// TIA Portal V20 export
FUNCTION_BLOCK "LER_EmOverviewHomeCondtion"   // FB182, LAD
// stored: IsIECCheckEnabled true, MemoryReserve 100, Namespace Unit1.Em2, SetENOAutomatically true
   VAR_INPUT
      maxPageCount : Int;
      unitStatus { ExternalAccessible := 'False'; ExternalVisible := 'False'; ExternalWritable := 'False'} : "LAF_typeUnitStatus";   // Current unit status o be used in this EM
   END_VAR
   VAR_IN_OUT
      moduleInterface : "LER_typeEmOverviewHomeCondition";
   END_VAR
   VAR
      statButtonPressedOld : Array[0..1] of Bool;
      statLampControl { ExternalAccessible := 'False'; ExternalVisible := 'False'; ExternalWritable := 'False'} : Bool;
      statPulse { ExternalAccessible := 'False'; ExternalVisible := 'False'; ExternalWritable := 'False'} : Bool;
   END_VAR
   VAR_TEMP
      tempLampOff : Array[0..13] of Bool;
   END_VAR
   VAR_TEMP   // added for the SCL form of the ladder/FBD networks
      _w1 : Bool;
      _w2 : Bool;
   END_VAR
BEGIN

REGION Network 1: Page Index Control
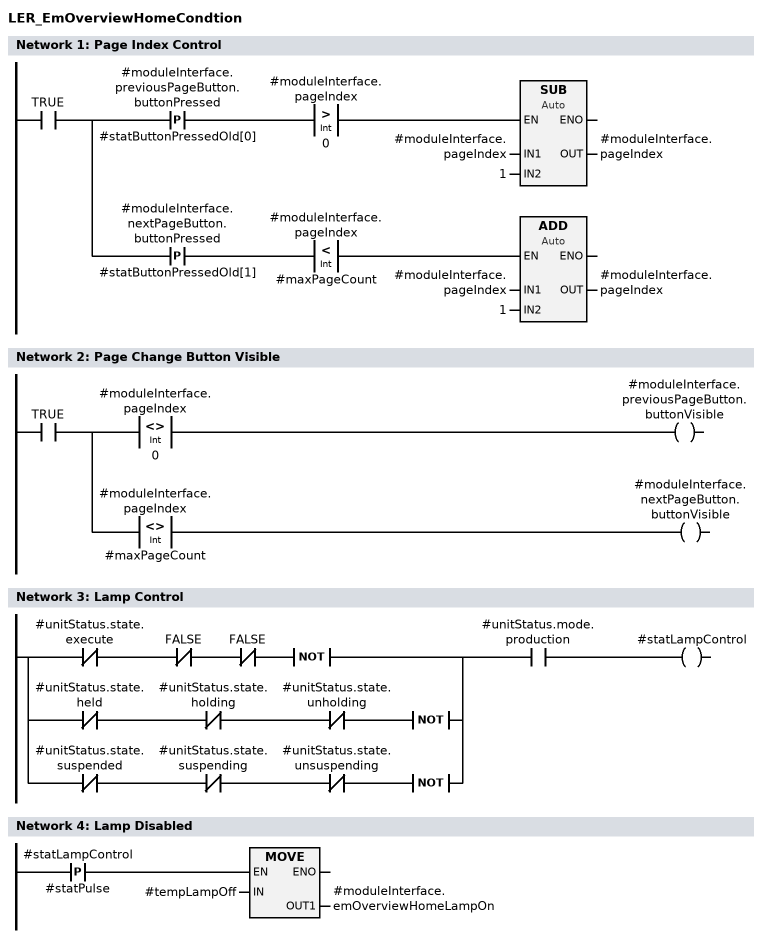
   RUNG wire#powerrail
      Contact( TRUE )
      wire#w1
      P_Contact(operand := #moduleInterface.previousPageButton.buttonPressed, bit := #statButtonPressedOld[0])
      { S7_Templates := "SrcType := Int" } GT_Contact(in1 := #moduleInterface.pageIndex, in2 := 0)
      Sub(in1 := #moduleInterface.pageIndex, in2 := 1, out => #moduleInterface.pageIndex)
   END_RUNG
   RUNG wire#w1
      P_Contact(operand := #moduleInterface.nextPageButton.buttonPressed, bit := #statButtonPressedOld[1])
      { S7_Templates := "SrcType := Int" } LT_Contact(in1 := #moduleInterface.pageIndex, in2 := #maxPageCount)
      Add(in1 := #moduleInterface.pageIndex, in2 := 1, out => #moduleInterface.pageIndex)
   END_RUNG
   // the same network as SCL:
   #_w1 := TRUE AND #moduleInterface.previousPageButton.buttonPressed AND NOT #statButtonPressedOld[0];   // rising edge of #moduleInterface.previousPageButton.buttonPressed
   #statButtonPressedOld[0] := #moduleInterface.previousPageButton.buttonPressed;
   IF #_w1 AND (#moduleInterface.pageIndex > 0) THEN
       #moduleInterface.pageIndex := #moduleInterface.pageIndex - 1;
   END_IF;
   #_w2 := TRUE AND #moduleInterface.nextPageButton.buttonPressed AND NOT #statButtonPressedOld[1];   // rising edge of #moduleInterface.nextPageButton.buttonPressed
   #statButtonPressedOld[1] := #moduleInterface.nextPageButton.buttonPressed;
   IF #_w2 AND (#moduleInterface.pageIndex < #maxPageCount) THEN
       #moduleInterface.pageIndex := #moduleInterface.pageIndex + 1;
   END_IF;
END_REGION

REGION Network 2: Page Change Button Visible
   RUNG wire#powerrail
      Contact( TRUE )
      wire#w1
      { S7_Templates := "SrcType := Int" } NE_Contact(in1 := #moduleInterface.pageIndex, in2 := 0)
      Coil( #moduleInterface.previousPageButton.buttonVisible )
   END_RUNG
   RUNG wire#w1
      { S7_Templates := "SrcType := Int" } NE_Contact(in1 := #moduleInterface.pageIndex, in2 := #maxPageCount)
      Coil( #moduleInterface.nextPageButton.buttonVisible )
   END_RUNG
   // the same network as SCL:
   #moduleInterface.previousPageButton.buttonVisible := TRUE AND (#moduleInterface.pageIndex <> 0);
   #moduleInterface.nextPageButton.buttonVisible := TRUE AND (#moduleInterface.pageIndex <> #maxPageCount);
END_REGION

REGION Network 3: Lamp Control
   RUNG wire#powerrail
      I_Contact( #unitStatus.state.execute )
      I_Contact( FALSE )
      I_Contact( FALSE )
      Not()
      wire#w1
      Contact( #unitStatus.mode.production )
      Coil( #statLampControl )
   END_RUNG
   RUNG wire#powerrail
      I_Contact( #unitStatus.state.held )
      I_Contact( #unitStatus.state.holding )
      I_Contact( #unitStatus.state.unholding )
      Not()
   END_RUNG wire#w1
   RUNG wire#powerrail
      I_Contact( #unitStatus.state.suspended )
      I_Contact( #unitStatus.state.suspending )
      I_Contact( #unitStatus.state.unsuspending )
      Not()
   END_RUNG wire#w1
   // the same network as SCL:
   #statLampControl := (NOT (NOT #unitStatus.state.execute AND NOT FALSE AND NOT FALSE) OR NOT (NOT #unitStatus.state.held AND NOT #unitStatus.state.holding AND NOT #unitStatus.state.unholding) OR NOT (NOT #unitStatus.state.suspended AND NOT #unitStatus.state.suspending AND NOT #unitStatus.state.unsuspending)) AND #unitStatus.mode.production;
END_REGION

REGION Network 4: Lamp Disabled
   RUNG wire#powerrail
      P_Contact(operand := #statLampControl, bit := #statPulse)
      Move(in := #tempLampOff, out1 => #moduleInterface.emOverviewHomeLampOn)
   END_RUNG
   // the same network as SCL:
   #_w1 := #statLampControl AND NOT #statPulse;   // rising edge of #statLampControl
   #statPulse := #statLampControl;
   IF #_w1 THEN #moduleInterface.emOverviewHomeLampOn := #tempLampOff; END_IF;
END_REGION

REGION Network 5 (SCL): Page Index 0 Mapping
   IF #moduleInterface.pageIndex = 0 THEN
     #moduleInterface.emOverviewTitle := WSTRING#'P&P Left Homed Condition 1';
     #moduleInterface.emOverviewCmName[0] := WSTRING#'Softcam Jelly Roll Out P&P Left Axis X';
     #moduleInterface.emOverviewCmName[1] := WSTRING#'Softcam Jelly Roll Out P&P Left Axis Z';
     #moduleInterface.emOverviewCmName[2] := WSTRING#'Jelly Roll Out P&P Left Jelly Roll Detect';
     #moduleInterface.emOverviewCmName[3] := WSTRING#'Jelly Roll Out P&P Left Clamp ';
     #moduleInterface.emOverviewCmName[4] := WSTRING#'Spare';
     #moduleInterface.emOverviewCmName[5] := WSTRING#'Spare';
     #moduleInterface.emOverviewCmName[6] := WSTRING#'Spare';
     #moduleInterface.emOverviewCmName[7] := WSTRING#'Spare';
     #moduleInterface.emOverviewCmName[8] := WSTRING#'Spare';
     #moduleInterface.emOverviewCmName[9] := WSTRING#'Spare';
     #moduleInterface.emOverviewCmName[10] := WSTRING#'Spare';
     #moduleInterface.emOverviewCmName[11] := WSTRING#'Spare';
     #moduleInterface.emOverviewCmName[12] := WSTRING#'Spare';
     #moduleInterface.emOverviewCmName[13] := WSTRING#'Spare';
     #moduleInterface.emOverviewCmPositionName[0] := WSTRING#'Wait Position';
     #moduleInterface.emOverviewCmPositionName[1] := WSTRING#'Wait Position';
     #moduleInterface.emOverviewCmPositionName[2] := WSTRING#'Not Detect';
     #moduleInterface.emOverviewCmPositionName[3] := WSTRING#'Open';
     #moduleInterface.emOverviewCmPositionName[4] := WSTRING#'Spare';
     #moduleInterface.emOverviewCmPositionName[5] := WSTRING#'Spare';
     #moduleInterface.emOverviewCmPositionName[6] := WSTRING#'Spare';
     #moduleInterface.emOverviewCmPositionName[7] := WSTRING#'Spare';
     #moduleInterface.emOverviewCmPositionName[8] := WSTRING#'Spare';
     #moduleInterface.emOverviewCmPositionName[9] := WSTRING#'Spare';
     #moduleInterface.emOverviewCmPositionName[10] := WSTRING#'Spare';
     #moduleInterface.emOverviewCmPositionName[11] := WSTRING#'Spare';
     #moduleInterface.emOverviewCmPositionName[12] := WSTRING#'Spare';
     #moduleInterface.emOverviewCmPositionName[13] := WSTRING#'Spare';

     IF NOT #statLampControl THEN
         #moduleInterface.emOverviewHomeLampOn[0] := "Unit1.Em2.ControlNodes".cm.softcam.jrOutPnPLeftAxisX.pos00_wait.inPos;
         #moduleInterface.emOverviewHomeLampOn[1] := "Unit1.Em2.ControlNodes".cm.softcam.jrOutPnPLeftAxisZ.pos00_wait.inPos;
         #moduleInterface.emOverviewHomeLampOn[2] := NOT "Unit1.Em2.ControlNodes".cmJROutPnPLeftJRDetect.monitoring.processValue;
         #moduleInterface.emOverviewHomeLampOn[3] := "Unit1.Em2.ControlNodes".cmJROutPnPLeftClampOpenClose.monitoring.inHomePos;
         #moduleInterface.emOverviewHomeLampOn[4] := FALSE;
         #moduleInterface.emOverviewHomeLampOn[5] := FALSE;
         #moduleInterface.emOverviewHomeLampOn[6] := FALSE;
         #moduleInterface.emOverviewHomeLampOn[7] := FALSE;
         #moduleInterface.emOverviewHomeLampOn[8] := FALSE;
         #moduleInterface.emOverviewHomeLampOn[9] := FALSE;
         #moduleInterface.emOverviewHomeLampOn[10] := FALSE;
         #moduleInterface.emOverviewHomeLampOn[11] := FALSE;
         #moduleInterface.emOverviewHomeLampOn[12] := FALSE;
         #moduleInterface.emOverviewHomeLampOn[13] := FALSE;
     END_IF;

   END_IF;
END_REGION

REGION Network 6 (SCL): Page Index 1 Mapping
   IF #moduleInterface.pageIndex = 1 THEN
       #moduleInterface.emOverviewTitle := WSTRING#'P&P Left Homed Condition 2';
     #moduleInterface.emOverviewCmName[0] := WSTRING#'Softcam Jelly Roll Out P&P Left Axis X';
     #moduleInterface.emOverviewCmName[1] := WSTRING#'Softcam Jelly Roll Out P&P Left Axis Z';
     #moduleInterface.emOverviewCmName[2] := WSTRING#'Jelly Roll Out P&P Left Jelly Roll Detect';
     #moduleInterface.emOverviewCmName[3] := WSTRING#'Jelly Roll Out P&P Left Clamp ';
     #moduleInterface.emOverviewCmName[4] := WSTRING#'Spare';
     #moduleInterface.emOverviewCmName[5] := WSTRING#'Spare';
     #moduleInterface.emOverviewCmName[6] := WSTRING#'Spare';
     #moduleInterface.emOverviewCmName[7] := WSTRING#'Spare';
     #moduleInterface.emOverviewCmName[8] := WSTRING#'Spare';
     #moduleInterface.emOverviewCmName[9] := WSTRING#'Spare';
     #moduleInterface.emOverviewCmName[10] := WSTRING#'Spare';
     #moduleInterface.emOverviewCmName[11] := WSTRING#'Spare';
     #moduleInterface.emOverviewCmName[12] := WSTRING#'Spare';
     #moduleInterface.emOverviewCmName[13] := WSTRING#'Spare';
     #moduleInterface.emOverviewCmPositionName[0] := WSTRING#'Wait Position';
     #moduleInterface.emOverviewCmPositionName[1] := WSTRING#'Wait Position';
     #moduleInterface.emOverviewCmPositionName[2] := WSTRING#'Detect';
     #moduleInterface.emOverviewCmPositionName[3] := WSTRING#'Close';
     #moduleInterface.emOverviewCmPositionName[4] := WSTRING#'Spare';
     #moduleInterface.emOverviewCmPositionName[5] := WSTRING#'Spare';
     #moduleInterface.emOverviewCmPositionName[6] := WSTRING#'Spare';
     #moduleInterface.emOverviewCmPositionName[7] := WSTRING#'Spare';
     #moduleInterface.emOverviewCmPositionName[8] := WSTRING#'Spare';
     #moduleInterface.emOverviewCmPositionName[9] := WSTRING#'Spare';
     #moduleInterface.emOverviewCmPositionName[10] := WSTRING#'Spare';
     #moduleInterface.emOverviewCmPositionName[11] := WSTRING#'Spare';
     #moduleInterface.emOverviewCmPositionName[12] := WSTRING#'Spare';
     #moduleInterface.emOverviewCmPositionName[13] := WSTRING#'Spare';

     IF NOT #statLampControl THEN
         #moduleInterface.emOverviewHomeLampOn[0] := "Unit1.Em2.ControlNodes".cm.softcam.jrOutPnPLeftAxisX.pos00_wait.inPos;
         #moduleInterface.emOverviewHomeLampOn[1] := "Unit1.Em2.ControlNodes".cm.softcam.jrOutPnPLeftAxisZ.pos00_wait.inPos;
         #moduleInterface.emOverviewHomeLampOn[2] := "Unit1.Em2.ControlNodes".cmJROutPnPLeftJRDetect.monitoring.processValue;
         #moduleInterface.emOverviewHomeLampOn[3] := "Unit1.Em2.ControlNodes".cmJROutPnPLeftClampOpenClose.monitoring.inWorkPos;
         #moduleInterface.emOverviewHomeLampOn[4] := FALSE;
         #moduleInterface.emOverviewHomeLampOn[5] := FALSE;
         #moduleInterface.emOverviewHomeLampOn[6] := FALSE;
         #moduleInterface.emOverviewHomeLampOn[7] := FALSE;
         #moduleInterface.emOverviewHomeLampOn[8] := FALSE;
         #moduleInterface.emOverviewHomeLampOn[9] := FALSE;
         #moduleInterface.emOverviewHomeLampOn[10] := FALSE;
         #moduleInterface.emOverviewHomeLampOn[11] := FALSE;
         #moduleInterface.emOverviewHomeLampOn[12] := FALSE;
         #moduleInterface.emOverviewHomeLampOn[13] := FALSE;
     END_IF;

   END_IF;
END_REGION

REGION Network 7 (SCL): Page Index 2 Mapping
   IF #moduleInterface.pageIndex = 2 THEN
       #moduleInterface.emOverviewTitle := WSTRING#'P&P Right Homed Condition 1';
     #moduleInterface.emOverviewCmName[0] := WSTRING#'Softcam Jelly Roll Out P&P Right Axis X';
     #moduleInterface.emOverviewCmName[1] := WSTRING#'Softcam Jelly Roll Out P&P Right Axis Z';
     #moduleInterface.emOverviewCmName[2] := WSTRING#'Jelly Roll Out P&P Right Jelly Roll Detect';
     #moduleInterface.emOverviewCmName[3] := WSTRING#'Jelly Roll Out P&P Right Clamp ';
     #moduleInterface.emOverviewCmName[4] := WSTRING#'Spare';
     #moduleInterface.emOverviewCmName[5] := WSTRING#'Spare';
     #moduleInterface.emOverviewCmName[6] := WSTRING#'Spare';
     #moduleInterface.emOverviewCmName[7] := WSTRING#'Spare';
     #moduleInterface.emOverviewCmName[8] := WSTRING#'Spare';
     #moduleInterface.emOverviewCmName[9] := WSTRING#'Spare';
     #moduleInterface.emOverviewCmName[10] := WSTRING#'Spare';
     #moduleInterface.emOverviewCmName[11] := WSTRING#'Spare';
     #moduleInterface.emOverviewCmName[12] := WSTRING#'Spare';
     #moduleInterface.emOverviewCmName[13] := WSTRING#'Spare';
     #moduleInterface.emOverviewCmPositionName[0] := WSTRING#'Wait Position';
     #moduleInterface.emOverviewCmPositionName[1] := WSTRING#'Wait Position';
     #moduleInterface.emOverviewCmPositionName[2] := WSTRING#'Not Detect';
     #moduleInterface.emOverviewCmPositionName[3] := WSTRING#'Open';
     #moduleInterface.emOverviewCmPositionName[4] := WSTRING#'Spare';
     #moduleInterface.emOverviewCmPositionName[5] := WSTRING#'Spare';
     #moduleInterface.emOverviewCmPositionName[6] := WSTRING#'Spare';
     #moduleInterface.emOverviewCmPositionName[7] := WSTRING#'Spare';
     #moduleInterface.emOverviewCmPositionName[8] := WSTRING#'Spare';
     #moduleInterface.emOverviewCmPositionName[9] := WSTRING#'Spare';
     #moduleInterface.emOverviewCmPositionName[10] := WSTRING#'Spare';
     #moduleInterface.emOverviewCmPositionName[11] := WSTRING#'Spare';
     #moduleInterface.emOverviewCmPositionName[12] := WSTRING#'Spare';
     #moduleInterface.emOverviewCmPositionName[13] := WSTRING#'Spare';

     IF NOT #statLampControl THEN
         #moduleInterface.emOverviewHomeLampOn[0] := "Unit1.Em2.ControlNodes".cm.softcam.jrOutPnPRightAxisX.pos00_wait.inPos;
         #moduleInterface.emOverviewHomeLampOn[1] := "Unit1.Em2.ControlNodes".cm.softcam.jrOutPnPRightAxisZ.pos00_wait.inPos;
         #moduleInterface.emOverviewHomeLampOn[2] := NOT "Unit1.Em2.ControlNodes".cmJROutPnPRightJRDetect.monitoring.processValue;
         #moduleInterface.emOverviewHomeLampOn[3] := "Unit1.Em2.ControlNodes".cmJROutPnPRightClampOpenClose.monitoring.inHomePos;
         #moduleInterface.emOverviewHomeLampOn[4] := FALSE;
         #moduleInterface.emOverviewHomeLampOn[5] := FALSE;
         #moduleInterface.emOverviewHomeLampOn[6] := FALSE;
         #moduleInterface.emOverviewHomeLampOn[7] := FALSE;
         #moduleInterface.emOverviewHomeLampOn[8] := FALSE;
         #moduleInterface.emOverviewHomeLampOn[9] := FALSE;
         #moduleInterface.emOverviewHomeLampOn[10] := FALSE;
         #moduleInterface.emOverviewHomeLampOn[11] := FALSE;
         #moduleInterface.emOverviewHomeLampOn[12] := FALSE;
         #moduleInterface.emOverviewHomeLampOn[13] := FALSE;
     END_IF;

   END_IF;
END_REGION

REGION Network 8 (SCL): Page Index 3 Mapping
   IF #moduleInterface.pageIndex = 3 THEN
       #moduleInterface.emOverviewTitle := WSTRING#'P&P Right Homed Condition 2';
     #moduleInterface.emOverviewCmName[0] := WSTRING#'Softcam Jelly Roll Out P&P Right Axis X';
     #moduleInterface.emOverviewCmName[1] := WSTRING#'Softcam Jelly Roll Out P&P Right Axis Z';
     #moduleInterface.emOverviewCmName[2] := WSTRING#'Jelly Roll Out P&P Right Jelly Roll Detect';
     #moduleInterface.emOverviewCmName[3] := WSTRING#'Jelly Roll Out P&P Right Clamp ';
     #moduleInterface.emOverviewCmName[4] := WSTRING#'Spare';
     #moduleInterface.emOverviewCmName[5] := WSTRING#'Spare';
     #moduleInterface.emOverviewCmName[6] := WSTRING#'Spare';
     #moduleInterface.emOverviewCmName[7] := WSTRING#'Spare';
     #moduleInterface.emOverviewCmName[8] := WSTRING#'Spare';
     #moduleInterface.emOverviewCmName[9] := WSTRING#'Spare';
     #moduleInterface.emOverviewCmName[10] := WSTRING#'Spare';
     #moduleInterface.emOverviewCmName[11] := WSTRING#'Spare';
     #moduleInterface.emOverviewCmName[12] := WSTRING#'Spare';
     #moduleInterface.emOverviewCmName[13] := WSTRING#'Spare';
     #moduleInterface.emOverviewCmPositionName[0] := WSTRING#'Wait Position';
     #moduleInterface.emOverviewCmPositionName[1] := WSTRING#'Wait Position';
     #moduleInterface.emOverviewCmPositionName[2] := WSTRING#'Detect';
     #moduleInterface.emOverviewCmPositionName[3] := WSTRING#'Close';
     #moduleInterface.emOverviewCmPositionName[4] := WSTRING#'Spare';
     #moduleInterface.emOverviewCmPositionName[5] := WSTRING#'Spare';
     #moduleInterface.emOverviewCmPositionName[6] := WSTRING#'Spare';
     #moduleInterface.emOverviewCmPositionName[7] := WSTRING#'Spare';
     #moduleInterface.emOverviewCmPositionName[8] := WSTRING#'Spare';
     #moduleInterface.emOverviewCmPositionName[9] := WSTRING#'Spare';
     #moduleInterface.emOverviewCmPositionName[10] := WSTRING#'Spare';
     #moduleInterface.emOverviewCmPositionName[11] := WSTRING#'Spare';
     #moduleInterface.emOverviewCmPositionName[12] := WSTRING#'Spare';
     #moduleInterface.emOverviewCmPositionName[13] := WSTRING#'Spare';

     IF NOT #statLampControl THEN
         #moduleInterface.emOverviewHomeLampOn[0] := "Unit1.Em2.ControlNodes".cm.softcam.jrOutPnPRightAxisX.pos00_wait.inPos;
         #moduleInterface.emOverviewHomeLampOn[1] := "Unit1.Em2.ControlNodes".cm.softcam.jrOutPnPRightAxisZ.pos00_wait.inPos;
         #moduleInterface.emOverviewHomeLampOn[2] := "Unit1.Em2.ControlNodes".cmJROutPnPRightJRDetect.monitoring.processValue;
         #moduleInterface.emOverviewHomeLampOn[3] := "Unit1.Em2.ControlNodes".cmJROutPnPRightClampOpenClose.monitoring.inWorkPos;
         #moduleInterface.emOverviewHomeLampOn[4] := FALSE;
         #moduleInterface.emOverviewHomeLampOn[5] := FALSE;
         #moduleInterface.emOverviewHomeLampOn[6] := FALSE;
         #moduleInterface.emOverviewHomeLampOn[7] := FALSE;
         #moduleInterface.emOverviewHomeLampOn[8] := FALSE;
         #moduleInterface.emOverviewHomeLampOn[9] := FALSE;
         #moduleInterface.emOverviewHomeLampOn[10] := FALSE;
         #moduleInterface.emOverviewHomeLampOn[11] := FALSE;
         #moduleInterface.emOverviewHomeLampOn[12] := FALSE;
         #moduleInterface.emOverviewHomeLampOn[13] := FALSE;
     END_IF;

   END_IF;
END_REGION
END_FUNCTION_BLOCK
